// TIA Portal V15.1 export
// export: Created 2026-01-15T16:29:42.8583456Z, ExportSetting WithDefaults, WithReadOnly, DisplayName Totally Integrated Automation Portal, DisplayVersion V15.1 Update 8, DisplayName TIA Portal Openness, DisplayVersion V15.1 Update 8, DisplayName STEP 7 Professional, DisplayVersion V15.1 Update 8, DisplayName WinCC Advanced, DisplayVersion V15.1 Update 8
DATA_BLOCK "6.3.WWAT1"   // DB609
{ S7_Optimized_Access := 'TRUE' }
VERSION : 0.1
// stored: AutoNumber false, CodeModifiedDate 2026-01-15T16:25:51.1061526Z, CompileDate 2026-01-15T16:25:51.1117172Z, CreationDate 2026-01-15T16:22:49.8270549Z, DBAccessibleFromOPCUA true, DownloadWithoutReinit false, InstanceOfName 6.WEIGHT_HANDLING, InstanceOfNumber 6, InstanceOfType FB, InterfaceModifiedDate 2023-12-29T17:39:18.5236469Z, IsConsistent true, IsKnowHowProtected false, IsRetainMemResEnabled false, MemoryReserve 100, ModifiedDate 2026-01-15T16:25:51.1061526Z, ParameterModified 2023-11-29T03:49:57.2782849Z, StructureModified 2023-12-29T17:39:18.5236469Z, UDAEnableTagReadback false
"6.WEIGHT_HANDLING"
   // VAR_INPUT
   //    W_IN { ExternalAccessible := 'False'; ExternalVisible := 'False'; ExternalWritable := 'False'} : Real;
   //    WR_IN : Real;
   //    PV_IN1 : Real;
   //    PV_IN2 : Real;
   //    PV_IN3 : Real;
   //    PV_IN4 : Real;
   //    PV_IN5 : Real;
   //    PV_IN6 : Real;
   //    SV_IN1 : Real;
   //    SV_IN2 : Real;
   //    SV_IN3 : Real;
   //    SV_IN4 : Real;
   //    SV_IN5 : Real;
   //    SV_IN6 : Real;
   //    RUN_1 { ExternalAccessible := 'False'; ExternalVisible := 'False'; ExternalWritable := 'False'} : Bool;
   //    RUN_2 { ExternalAccessible := 'False'; ExternalVisible := 'False'; ExternalWritable := 'False'} : Bool;
   //    RUN_3 { ExternalAccessible := 'False'; ExternalVisible := 'False'; ExternalWritable := 'False'} : Bool;
   //    RUN_4 { ExternalAccessible := 'False'; ExternalVisible := 'False'; ExternalWritable := 'False'} : Bool;
   //    RUN_5 { ExternalAccessible := 'False'; ExternalVisible := 'False'; ExternalWritable := 'False'} : Bool;
   //    RUN_6 { ExternalAccessible := 'False'; ExternalVisible := 'False'; ExternalWritable := 'False'} : Bool;
   //    EMTY { ExternalAccessible := 'False'; ExternalVisible := 'False'; ExternalWritable := 'False'} : Bool;
   // END_VAR
   // VAR_OUTPUT
   //    W_OUT1 { ExternalAccessible := 'False'; ExternalVisible := 'False'; ExternalWritable := 'False'} : Real;
   //    W_OUT2 { ExternalAccessible := 'False'; ExternalVisible := 'False'; ExternalWritable := 'False'} : Real;
   //    W_OUT3 { ExternalAccessible := 'False'; ExternalVisible := 'False'; ExternalWritable := 'False'} : Real;
   //    W_OUT4 { ExternalAccessible := 'False'; ExternalVisible := 'False'; ExternalWritable := 'False'} : Real;
   //    W_OUT5 { ExternalAccessible := 'False'; ExternalVisible := 'False'; ExternalWritable := 'False'} : Real;
   //    W_OUT6 { ExternalAccessible := 'False'; ExternalVisible := 'False'; ExternalWritable := 'False'} : Real;
   //    "%W_OUT" { ExternalAccessible := 'False'; ExternalVisible := 'False'; ExternalWritable := 'False'} : Real;
   // END_VAR
   // VAR RETAIN
   //    W_Star : Real;
   //    W_Temp : Real;
   // END_VAR
   // VAR
   //    P_RUN1 : Bool;
   //    P_RUN2 : Bool;
   //    P_RUN3 : Bool;
   //    P_RUN4 : Bool;
   //    P_RUN5 : Bool;
   //    P_RUN6 : Bool;
   //    N_RUN1 : Bool;
   //    N_RUN2 : Bool;
   //    N_RUN3 : Bool;
   //    N_RUN4 : Bool;
   //    N_RUN5 : Bool;
   //    N_RUN6 : Bool;
   // END_VAR
   // VAR RETAIN
   //    PV1 : Real;
   //    PV2 : Real;
   //    PV3 : Real;
   //    PV4 : Real;
   //    PV5 : Real;
   //    PV6 : Real;
   // END_VAR
BEGIN
END_DATA_BLOCK
